// SIMATIC S7-200 project (STEP 7-Micro/WIN), CPU 221 REL 01.10

ORGANIZATION_BLOCK MAIN:OB1
TITLE=这个项目包含CRC码计算和发送模块，实现工业自动化控制系统中通过Modbus RTU协议与变频器通信。
// 生成并发送读取命令以获取寄存器数据，控制设备包括变频器和PLC通信模块。
// 系统启动时，初始化发送数据区：数据长度设置为8字节，确保与实际数据匹配；变频器地址设为1，功能代码设为读取功能（16#03），两者需保持有效以便变频器正确识别；
// 寄存器地址高位和寄存器地址低位组成地址0x0065，指向目标寄存器；数据高位和数据低位指定读取3个寄存器的数据量。
// 特别地，数据长度需保持8字节以确保后续CRC计算的正确性，变频器地址需与实际地址一致以保证变频器响应，功能代码需为03以执行预期操作，寄存器地址高位和低位需形成有效地址以获取正确数据。
// 同时，CRC寄存器初始化为0xFFFF，循环指针指向数据长度，为后续计算做准备，这里循环指针需准确指向数据长度以基于正确数据进行计算。
// CRC计算过程从发送数据区开始，异或循环计数器驱动6次循环，处理每个字节，确保异或循环计数器达到6次以完整覆盖数据。
// 循环指针逐字节递增，确保覆盖所有数据，将当前字节存入异或数据字节，异或数据高位置0，组成异或操作寄存器与CRC寄存器异或。
// 对每个字节，右移次数计数器控制8次右移，CRC寄存器每次右移一位，最低位状态通过系统最低位标志检查最低位，若为1则与0xA001异或，需确保右移次数计数器达到8次以保证CRC结果准确。
// 计算完成后，CRC寄存器的低字节和高字节分别存入CRC低位和CRC高位，并按低位在前、高位在后的顺序附加到命令中，符合协议要求。
// 
// 
BEGIN
Network 1 // 网络标题// CRC初始化
// 网络注释
// 初始化CRC寄存器,设置发送区指针.
LD     SM0.0
R      M20.1, 1
MOVB   16#8, VB100           //数据长度
MOVB   16#1, VB101           //变频器地址
MOVB   16#3, VB102           //功能代码,读取.
MOVB   16#0, VB103           //寄存地址高位
MOVB   16#65, VB104          //寄存地址低位
MOVB   16#0, VB105           //数据高位
MOVB   16#3, VB106           //数据低位
MOVW   16#FFFF, VW350        //将CRC寄存器设置为FFFF.
MOVD   &VB100, VD54          //设定循环指针.
Network 2
// 设置异或循环次数,使循环指针加1;信息和CRC寄存器异或.
LD     SM0.0
FOR    VW50, +1, +6          //设置异或循环次数.
INCD   VD54                  //循环指针加1
MOVB   *VD54, VB201          //将需要异或的数据放入VB201,即VW200的低位.
MOVB   0, VB200              //将VW200的高位置0
XORW   VW200, VW350          //信息字符与CRC寄存器异或.
Network 3
// 设置右移次数,右移CRC寄存器内数据八次,且检查每次右移后CRC寄存器最低位的状态是否为1,是则和A001异或.
LD     SM0.0
FOR    VW52, +1, +8          //设置右移次数
SRW    VW350, 1              //CRC寄存器右移一位
MOVB   SMB1, VB58            //检查VW350最低位是否为1
ANDB   16#2, VB58
AB=    VB58, 2               //是
XORW   16#A001, VW350        //和HEX的A001进行异或处理
Network 4
// 右移之FOR>>>>NEXT
NEXT                         //右移次数未到达时回FOR处,共八次
Network 5
//异或次数之FOR>>>>>>NEXT
NEXT                         //数据异或次数未达到时回FOR,共六次.
Network 6
LD     SM0.0
MOVB   VB351, VB107          //CRC数据低位
MOVB   VB350, VB108          //CRC数据高位
CALL   发送_READ:SBR0
END_ORGANIZATION_BLOCK
